	PROC rRUNSIDE1A100()
		MoveJ [[895.91,925.45,959.23],[0.222593,0.0151737,0.948305,-0.225698],[0,-1,0,0],[9E+09,9E+09,9E+09,9E+09,9E+09,9E+09]], vmax, z50, tWeldGun;
		MoveJ [[1169.38,1081.61,325.39],[0.296115,-0.947077,-0.052822,0.112127],[0,-2,0,1],[9E+09,9E+09,9E+09,9E+09,9E+09,9E+09]], vmax, z50, tWeldGun;
		MoveL [[1189.01,1078.57,4.64],[0.333702,-0.921867,0.118424,-0.157418],[0,-2,-1,1],[9E+09,9E+09,9E+09,9E+09,9E+09,9E+09]], v1000, z50, tWeldGun;
		ArcLStart [[1185.61,1080.58,-9.86],[0.333643,-0.921896,0.118528,-0.157299],[0,-2,-1,1],[9E+09,9E+09,9E+09,9E+09,9E+09,9E+09]], v10, seam13, weld13\Weave:=weave1, fine, tWeldGun;
		ArcLEnd [[1153.22,1080.55,-9.89],[0.333626,-0.921901,0.118526,-0.157301],[0,-2,-1,1],[9E+09,9E+09,9E+09,9E+09,9E+09,9E+09]], v10, seam13, weld13\Weave:=weave1, fine, tWeldGun;
		MoveL [[1157.55,1079.96,5.67],[0.333709,-0.921874,0.118398,-0.157383],[0,-2,-1,1],[9E+09,9E+09,9E+09,9E+09,9E+09,9E+09]], vmax, z5, tWeldGun;
		MoveL [[864.56,1073.01,5.26],[0.379695,-0.916748,-0.042496,0.116617],[0,-2,-1,1],[9E+09,9E+09,9E+09,9E+09,9E+09,9E+09]], vmax, z5, tWeldGun;
		ArcLStart [[862.19,1074.19,-3.35],[0.379691,-0.916749,-0.0424859,0.116625],[0,-2,-1,1],[9E+09,9E+09,9E+09,9E+09,9E+09,9E+09]], v10, seam13, weld13\Weave:=weave1, fine, tWeldGun;
		ArcLEnd [[831.24,1074.23,-3.33],[0.379713,-0.916742,-0.0424399,0.116624],[0,-2,-1,1],[9E+09,9E+09,9E+09,9E+09,9E+09,9E+09]], v10, seam13, weld13\Weave:=weave1, fine, tWeldGun;
		MoveL [[834.56,1075.21,12.06],[0.379682,-0.916754,-0.0425092,0.116603],[0,-2,-1,1],[9E+09,9E+09,9E+09,9E+09,9E+09,9E+09]], vmax, z5, tWeldGun;
		MoveL [[172.30,1074.14,5.27],[0.379642,-0.916784,-0.0424626,0.11652],[0,-2,-1,1],[9E+09,9E+09,9E+09,9E+09,9E+09,9E+09]], vmax, z5, tWeldGun;
		ArcLStart [[172.45,1077.16,-3.73],[0.37965,-0.916783,-0.042437,0.116513],[0,-2,-1,1],[9E+09,9E+09,9E+09,9E+09,9E+09,9E+09]], v10, seam13, weld13\Weave:=weave1, fine, tWeldGun;
		ArcLEnd [[141.11,1075.63,-6.35],[0.394237,-0.896713,-0.191368,0.0621412],[0,-2,-1,1],[9E+09,9E+09,9E+09,9E+09,9E+09,9E+09]], v10, seam13, weld13\Weave:=weave1, fine, tWeldGun;
		MoveL [[141.10,1062.84,1.66],[0.394214,-0.896726,-0.191336,0.0621991],[0,-2,-1,1],[9E+09,9E+09,9E+09,9E+09,9E+09,9E+09]], vmax, z5, tWeldGun;
		MoveL [[-144.86,1070.65,3.80],[0.337591,-0.932768,-0.0489574,0.116536],[0,-2,-1,1],[9E+09,9E+09,9E+09,9E+09,9E+09,9E+09]], vmax, z5, tWeldGun;
		ArcLStart [[-144.83,1077.50,-2.20],[0.337605,-0.932765,-0.048953,0.116519],[0,-2,-1,1],[9E+09,9E+09,9E+09,9E+09,9E+09,9E+09]], v10, seam13, weld13\Weave:=weave1, fine, tWeldGun;
		ArcLEnd [[-176.80,1077.27,-2.42],[0.337568,-0.932779,-0.0489017,0.116534],[0,-2,-1,1],[9E+09,9E+09,9E+09,9E+09,9E+09,9E+09]], v10, seam13, weld13\Weave:=weave1, fine, tWeldGun;
		SingArea\Wrist;
		MoveL [[-200.44,1085.42,415.26],[0.379667,-0.916774,-0.042596,0.116465],[0,-2,-1,1],[9E+09,9E+09,9E+09,9E+09,9E+09,9E+09]], vmax, z5, tWeldGun;
		MoveJ [[-173.57,559.75,42.74],[0.145109,0.845875,-0.418866,0.296634],[1,0,-1,0],[9E+09,9E+09,9E+09,9E+09,9E+09,9E+09]], vmax, z5, tWeldGun;
		MoveL [[-170.35,568.46,-5.16],[0.145203,0.845842,-0.418973,0.29653],[1,0,-1,0],[9E+09,9E+09,9E+09,9E+09,9E+09,9E+09]], vmax, z5, tWeldGun;
		ArcLStart [[-170.35,561.67,-11.54],[0.145203,0.845851,-0.418953,0.296532],[1,0,-1,0],[9E+09,9E+09,9E+09,9E+09,9E+09,9E+09]], v10, seam13, weld13\Weave:=weave1, fine, tWeldGun;
		ArcLEnd [[-141.78,561.68,-11.54],[0.145216,0.845844,-0.418977,0.296513],[1,0,-1,0],[9E+09,9E+09,9E+09,9E+09,9E+09,9E+09]], v10, seam13, weld13\Weave:=weave1, fine, tWeldGun;
		MoveL [[-135.50,566.77,5.60],[0.145085,0.84588,-0.41892,0.296555],[1,0,-1,0],[9E+09,9E+09,9E+09,9E+09,9E+09,9E+09]], vmax, z5, tWeldGun;
		MoveL [[151.70,563.89,2.38],[0.145279,0.845821,-0.418979,0.296543],[0,0,-1,0],[9E+09,9E+09,9E+09,9E+09,9E+09,9E+09]], vmax, z5, tWeldGun;
		ArcLStart [[147.91,561.67,-12.61],[0.145298,0.845824,-0.41896,0.296552],[0,0,-1,0],[9E+09,9E+09,9E+09,9E+09,9E+09,9E+09]], v10, seam13, weld13\Weave:=weave1, fine, tWeldGun;
		ArcLEnd [[179.68,561.61,-12.60],[0.145306,0.845823,-0.418965,0.296545],[0,0,-1,0],[9E+09,9E+09,9E+09,9E+09,9E+09,9E+09]], v10, seam13, weld13\Weave:=weave1, fine, tWeldGun;
		MoveL [[179.70,567.65,-1.58],[0.145437,0.845826,-0.418906,0.296553],[0,0,-1,0],[9E+09,9E+09,9E+09,9E+09,9E+09,9E+09]], vmax, z5, tWeldGun;
		MoveL [[838.33,565.65,0.78],[0.145096,0.845788,-0.419047,0.296632],[0,0,-2,0],[9E+09,9E+09,9E+09,9E+09,9E+09,9E+09]], vmax, z5, tWeldGun;
		ArcLStart [[837.91,559.63,-15.44],[0.14512,0.845784,-0.419056,0.29662],[0,0,-2,0],[9E+09,9E+09,9E+09,9E+09,9E+09,9E+09]], v10, seam13, weld13\Weave:=weave1, fine, tWeldGun;
		ArcLEnd [[868.85,559.41,-15.48],[0.145145,0.845802,-0.419023,0.296601],[0,0,-2,0],[9E+09,9E+09,9E+09,9E+09,9E+09,9E+09]], v10, seam13, weld13\Weave:=weave1, fine, tWeldGun;
		MoveL [[869.08,565.56,-7.05],[0.145032,0.845778,-0.419043,0.296696],[0,0,-2,0],[9E+09,9E+09,9E+09,9E+09,9E+09,9E+09]], vmax, z5, tWeldGun;
		MoveL [[1154.26,567.31,-2.43],[0.145055,0.845814,-0.419044,0.296583],[0,0,-2,0],[9E+09,9E+09,9E+09,9E+09,9E+09,9E+09]], vmax, z5, tWeldGun;
		ArcLStart [[1154.25,559.10,-16.64],[0.145066,0.845816,-0.419041,0.296576],[0,0,-2,0],[9E+09,9E+09,9E+09,9E+09,9E+09,9E+09]], v10, seam13, weld13\Weave:=weave1, fine, tWeldGun;
		ArcLEnd [[1186.24,558.29,-16.04],[0.145087,0.845809,-0.419057,0.296562],[0,0,-2,0],[9E+09,9E+09,9E+09,9E+09,9E+09,9E+09]], v10, seam13, weld13\Weave:=weave1, fine, tWeldGun;
		MoveL [[1189.43,560.09,663.81],[0.145007,0.845796,-0.418995,0.296726],[0,0,-2,0],[9E+09,9E+09,9E+09,9E+09,9E+09,9E+09]], vmax, z5, tWeldGun;
		MoveJ [[-229.23,1115.81,554.88],[0.237488,0.691166,-0.628837,0.265431],[1,-1,-4,0],[9E+09,9E+09,9E+09,9E+09,9E+09,9E+09]], vmax, z5, tWeldGun;
		MoveL [[-412.06,717.19,27.71],[0.270403,0.66951,-0.638814,0.265624],[1,0,-4,0],[9E+09,9E+09,9E+09,9E+09,9E+09,9E+09]], vmax, z5, tWeldGun;
		MoveL [[-413.84,720.92,-0.46],[0.249904,0.677081,-0.652542,0.230865],[1,-1,-4,0],[9E+09,9E+09,9E+09,9E+09,9E+09,9E+09]], vmax, z5, tWeldGun;
		ArcLStart [[-413.85,715.51,-6.45],[0.249932,0.67707,-0.652544,0.230859],[1,-1,-4,0],[9E+09,9E+09,9E+09,9E+09,9E+09,9E+09]], v5, seam13, weld13\Weave:=weave1, fine, tWeldGun;
		ArcLEnd [[-433.02,715.70,-6.65],[0.249921,0.677092,-0.652516,0.230888],[1,-1,-4,0],[9E+09,9E+09,9E+09,9E+09,9E+09,9E+09]], v5, seam13, weld13\Weave:=weave1, fine, tWeldGun;
		MoveL [[-433.02,721.69,79.27],[0.249938,0.677071,-0.652532,0.230886],[1,-1,-4,0],[9E+09,9E+09,9E+09,9E+09,9E+09,9E+09]], vmax, z5, tWeldGun;
		MoveL [[-1100.50,721.09,94.11],[0.270393,0.669535,-0.638788,0.265635],[1,-1,-4,0],[9E+09,9E+09,9E+09,9E+09,9E+09,9E+09]], vmax, z5, tWeldGun;
		MoveL [[-1103.19,722.45,8.00],[0.239603,0.681202,-0.652992,0.228379],[1,-1,-4,0],[9E+09,9E+09,9E+09,9E+09,9E+09,9E+09]], vmax, z5, tWeldGun;
		ArcLStart [[-1103.19,713.56,-5.56],[0.239599,0.681202,-0.652993,0.228381],[1,-1,-4,0],[9E+09,9E+09,9E+09,9E+09,9E+09,9E+09]], v5, seam13, weld13\Weave:=weave1, fine, tWeldGun;
		ArcLEnd [[-1123.14,713.55,-4.77],[0.239595,0.681192,-0.652991,0.228416],[1,-1,-4,0],[9E+09,9E+09,9E+09,9E+09,9E+09,9E+09]], v5, seam13, weld13\Weave:=weave1, fine, tWeldGun;
		MoveL [[-1124.97,712.38,115.49],[0.270384,0.669531,-0.638781,0.26567],[1,-1,-4,0],[9E+09,9E+09,9E+09,9E+09,9E+09,9E+09]], vmax, z5, tWeldGun;
		MoveJ [[-1119.62,941.62,98.59],[0.263153,-0.665669,-0.65042,-0.254146],[1,0,-2,0],[9E+09,9E+09,9E+09,9E+09,9E+09,9E+09]], vmax, z5, tWeldGun;
		MoveL [[-1103.53,941.47,2.67],[0.263185,-0.665692,-0.650383,-0.254147],[1,0,-2,0],[9E+09,9E+09,9E+09,9E+09,9E+09,9E+09]], vmax, z5, tWeldGun;
		ArcLStart [[-1102.50,948.16,-6.90],[0.245378,-0.666002,-0.671984,-0.211351],[1,0,-2,0],[9E+09,9E+09,9E+09,9E+09,9E+09,9E+09]], v5, seam13, weld13\Weave:=weave1, fine, tWeldGun;
		ArcL [[-1124.20,945.08,-8.53],[0.241268,-0.666756,-0.672776,-0.211185],[1,0,-2,0],[9E+09,9E+09,9E+09,9E+09,9E+09,9E+09]], v5, seam13, weld13\Weave:=weave1, z10, tWeldGun;
		ArcLEnd [[-1132.51,978.64,-7.54],[0.0250689,0.926224,0.0082503,0.376049],[1,0,-1,0],[9E+09,9E+09,9E+09,9E+09,9E+09,9E+09]], v5, seam13, weld13\Weave:=weave1, fine, tWeldGun;
		MoveL [[-1148.62,985.17,63.09],[0.0198579,0.898733,0.00249179,0.438039],[1,-1,-1,0],[9E+09,9E+09,9E+09,9E+09,9E+09,9E+09]], vmax, z5, tWeldGun;
		MoveL [[-1199.14,1157.80,50.93],[0.0198608,0.898743,0.00250084,0.43802],[1,-1,-1,0],[9E+09,9E+09,9E+09,9E+09,9E+09,9E+09]], vmax, z5, tWeldGun;
		MoveL [[-1195.49,1156.64,0.22],[0.0202314,0.914596,0.00160063,0.403859],[1,0,-1,0],[9E+09,9E+09,9E+09,9E+09,9E+09,9E+09]], vmax, z5, tWeldGun;
		ArcLStart [[-1192.13,1157.24,-7.56],[0.0202377,0.91461,0.00159549,0.403829],[1,0,-1,0],[9E+09,9E+09,9E+09,9E+09,9E+09,9E+09]], v5, seam13, weld13\Weave:=weave1, fine, tWeldGun;
		ArcL [[-1195.11,1177.16,-6.96],[0.0243873,0.92589,-0.000794778,0.377005],[1,0,-1,0],[9E+09,9E+09,9E+09,9E+09,9E+09,9E+09]], v5, seam13, weld13\Weave:=weave1, z10, tWeldGun;
		ArcLEnd [[-1166.64,1194.35,-4.47],[0.234917,0.673253,-0.666667,0.217024],[1,-1,0,0],[9E+09,9E+09,9E+09,9E+09,9E+09,9E+09]], v5, seam13, weld13\Weave:=weave1, fine, tWeldGun;
		MoveL [[-1164.13,1200.44,93.33],[0.251271,0.657126,-0.66952,0.23831],[1,-1,0,0],[9E+09,9E+09,9E+09,9E+09,9E+09,9E+09]], vmax, z5, tWeldGun;
		MoveJ [[-1176.39,1428.24,109.35],[0.303454,-0.641239,-0.63752,-0.300495],[1,-1,2,0],[9E+09,9E+09,9E+09,9E+09,9E+09,9E+09]], vmax, z5, tWeldGun;
		MoveL [[-1186.42,1420.24,9.09],[0.262683,-0.660481,-0.654281,-0.258224],[1,0,2,0],[9E+09,9E+09,9E+09,9E+09,9E+09,9E+09]], vmax, z5, tWeldGun;
		ArcLStart [[-1183.89,1427.01,-5.32],[0.262685,-0.660493,-0.654268,-0.258224],[1,0,2,0],[9E+09,9E+09,9E+09,9E+09,9E+09,9E+09]], v30, seam13, weld13\Weave:=weave1, fine, tWeldGun;
		ArcLEnd [[-1164.71,1427.19,-6.55],[0.262711,-0.66047,-0.654286,-0.258211],[1,0,2,0],[9E+09,9E+09,9E+09,9E+09,9E+09,9E+09]], v5, seam13, weld13\Weave:=weave1, fine, tWeldGun;
		MoveL [[-1165.10,1427.68,74.68],[0.262682,-0.660472,-0.654289,-0.258226],[1,0,2,0],[9E+09,9E+09,9E+09,9E+09,9E+09,9E+09]], vmax, z5, tWeldGun;
		MoveL [[-495.20,1424.53,122.41],[0.28862,-0.64963,-0.643265,-0.284411],[1,-1,2,0],[9E+09,9E+09,9E+09,9E+09,9E+09,9E+09]], vmax, z5, tWeldGun;
		MoveL [[-492.11,1424.64,-4.56],[0.230632,-0.671635,-0.668577,-0.220728],[1,0,2,0],[9E+09,9E+09,9E+09,9E+09,9E+09,9E+09]], vmax, z5, tWeldGun;
		ArcLStart [[-494.82,1430.84,-11.36],[0.230629,-0.671668,-0.668546,-0.220726],[1,0,2,0],[9E+09,9E+09,9E+09,9E+09,9E+09,9E+09]], v5, seam13, weld13\Weave:=weave1, fine, tWeldGun;
		ArcLEnd [[-475.00,1430.64,-11.57],[0.230621,-0.671683,-0.668534,-0.220724],[1,0,2,0],[9E+09,9E+09,9E+09,9E+09,9E+09,9E+09]], v5, seam13, weld13\Weave:=weave1, fine, tWeldGun;
		MoveL [[-474.63,1411.30,125.45],[0.288602,-0.649679,-0.643225,-0.284408],[1,-1,2,0],[9E+09,9E+09,9E+09,9E+09,9E+09,9E+09]], vmax, z5, tWeldGun;
		MoveJ [[-479.04,1241.31,118.19],[0.268582,0.650118,-0.664304,0.252806],[1,-1,0,0],[9E+09,9E+09,9E+09,9E+09,9E+09,9E+09]], vmax, z5, tWeldGun;
		MoveL [[-495.83,1201.80,-1.90],[0.268594,0.650121,-0.6643,0.252797],[1,-1,0,0],[9E+09,9E+09,9E+09,9E+09,9E+09,9E+09]], vmax, z5, tWeldGun;
		ArcLStart [[-494.84,1196.21,-9.49],[0.268603,0.650127,-0.664292,0.252793],[1,-1,0,0],[9E+09,9E+09,9E+09,9E+09,9E+09,9E+09]], v5, seam13, weld13\Weave:=weave1, fine, tWeldGun;
		ArcL [[-476.48,1196.50,-9.26],[0.268632,0.650097,-0.664312,0.252787],[1,-1,0,0],[9E+09,9E+09,9E+09,9E+09,9E+09,9E+09]], v5, seam13, weld13\Weave:=weave1, z10, tWeldGun;
		ArcLEnd [[-465.51,1166.36,-12.09],[0.390509,0.0535053,-0.919043,-0.000194166],[1,-1,1,0],[9E+09,9E+09,9E+09,9E+09,9E+09,9E+09]], v5, seam13, weld13\Weave:=weave1, fine, tWeldGun;
		MoveL [[-435.96,1164.94,59.58],[0.390502,0.0535497,-0.919044,-0.000186584],[1,-1,1,0],[9E+09,9E+09,9E+09,9E+09,9E+09,9E+09]], vmax, z5, tWeldGun;
		MoveL [[-398.53,986.99,7.96],[0.390518,0.0535228,-0.919039,-0.00018247],[1,-1,1,0],[9E+09,9E+09,9E+09,9E+09,9E+09,9E+09]], vmax, z5, tWeldGun;
		ArcLStart [[-404.11,986.56,-9.77],[0.390535,0.0535541,-0.919029,-0.000151074],[1,-1,1,0],[9E+09,9E+09,9E+09,9E+09,9E+09,9E+09]], v20, seam13, weld13\Weave:=weave1, fine, tWeldGun;
		ArcL [[-404.10,964.74,-9.51],[0.390566,0.0535448,-0.919017,-0.000185269],[1,-1,1,0],[9E+09,9E+09,9E+09,9E+09,9E+09,9E+09]], v5, seam13, weld13\Weave:=weave1, z10, tWeldGun;
		ArcLEnd [[-428.88,950.30,-8.06],[0.237036,-0.623338,-0.70044,-0.254259],[1,-1,2,0],[9E+09,9E+09,9E+09,9E+09,9E+09,9E+09]], v5, seam13, weld13\Weave:=weave1, fine, tWeldGun;
		MoveL [[-432.86,900.19,113.28],[0.289357,-0.647919,-0.645007,-0.283619],[1,-1,2,0],[9E+09,9E+09,9E+09,9E+09,9E+09,9E+09]], vmax, z5, tWeldGun;
		MoveJ [[276.57,1109.67,795.31],[0.28935,-0.647904,-0.645024,-0.283623],[0,0,1,0],[9E+09,9E+09,9E+09,9E+09,9E+09,9E+09]], vmax, z5, tWeldGun;
	ENDPROC
	PROC ProSkid200()
		MoveJ pSafeS1, vmax, fine, tWeldGun;
		MoveL [[-234.96,1621.92,-8.21],[0.194298,-0.276185,-0.910115,-0.24013],[1,-1,1,0],[9E+09,9E+09,9E+09,9E+09,9E+09,9E+09]], vmax, z50, tWeldGun;
		SingArea\Wrist;
		ArcLStart [[-265.19,1628.57,-38.88],[0.243445,-0.67037,-0.655025,-0.249563],[1,0,2,0],[9E+09,9E+09,9E+09,9E+09,9E+09,9E+09]], v40, seam13, weld13, fine, tWeldGun;
		ArcLEnd [[-257.54,1628.57,-38.88],[0.243445,-0.670369,-0.655025,-0.249565],[1,0,2,0],[9E+09,9E+09,9E+09,9E+09,9E+09,9E+09]], v10, seam13, weld13, fine, tWeldGun;
		MoveL [[-258.35,1618.76,-2.87],[0.243441,-0.670362,-0.655032,-0.24957],[1,0,2,0],[9E+09,9E+09,9E+09,9E+09,9E+09,9E+09]], vmax, z20, tWeldGun;
		MoveJ [[-252.87,717.22,166.31],[0.308554,0.634187,-0.646071,0.291883],[1,0,0,0],[9E+09,9E+09,9E+09,9E+09,9E+09,9E+09]], vmax, z20, tWeldGun;
		SingArea\Wrist;
		MoveL [[-273.06,697.08,-39.01],[0.289422,0.639754,-0.670959,0.238254],[1,0,0,0],[9E+09,9E+09,9E+09,9E+09,9E+09,9E+09]], vmax, z20, tWeldGun;
		ArcLStart [[-273.06,687.07,-45.02],[0.289425,0.639748,-0.670962,0.238258],[1,0,0,0],[9E+09,9E+09,9E+09,9E+09,9E+09,9E+09]], v10, seam13, weld13, fine, tWeldGun;
		ArcLEnd [[-266.46,687.08,-45.02],[0.289425,0.63975,-0.67096,0.238257],[1,0,0,0],[9E+09,9E+09,9E+09,9E+09,9E+09,9E+09]], v10, seam13, weld13, fine, tWeldGun;
		MoveL [[-265.17,697.65,3.08],[0.289425,0.639755,-0.670954,0.238258],[1,0,0,0],[9E+09,9E+09,9E+09,9E+09,9E+09,9E+09]], vmax, z20, tWeldGun;
		MoveJ [[1363.12,672.47,163.81],[0.230647,0.704641,-0.28697,0.606574],[0,-1,-1,0],[9E+09,9E+09,9E+09,9E+09,9E+09,9E+09]], vmax, z20, tWeldGun;
		MoveL [[1363.13,672.48,-59.34],[0.230635,0.704646,-0.28697,0.606573],[0,-1,-1,0],[9E+09,9E+09,9E+09,9E+09,9E+09,9E+09]], vmax, z20, tWeldGun;
		ArcLStart [[1395.10,665.67,-59.36],[0.230647,0.704646,-0.286968,0.606569],[0,-1,-1,0],[9E+09,9E+09,9E+09,9E+09,9E+09,9E+09]], v10, seam13, weld13, fine, tWeldGun;
		ArcLEnd [[1393.21,666.82,-105.76],[0.230653,0.704647,-0.286991,0.606554],[0,-1,-1,0],[9E+09,9E+09,9E+09,9E+09,9E+09,9E+09]], v10, seam13, weld13, fine, tWeldGun;
		MoveL [[1360.51,678.95,-105.76],[0.230657,0.704646,-0.286998,0.60655],[0,-1,-1,0],[9E+09,9E+09,9E+09,9E+09,9E+09,9E+09]], vmax, z20, tWeldGun;
		MoveJ [[1360.48,679.11,200.26],[0.227916,0.703475,-0.290109,0.607465],[0,-1,-1,0],[9E+09,9E+09,9E+09,9E+09,9E+09,9E+09]], vmax, z20, tWeldGun;
		MoveJ [[1372.60,1612.03,89.61],[0.238536,-0.688587,-0.26592,-0.631059],[0,-1,-2,0],[9E+09,9E+09,9E+09,9E+09,9E+09,9E+09]], vmax, z20, tWeldGun;
		MoveL [[1372.62,1612.07,-51.09],[0.238534,-0.68856,-0.265944,-0.631079],[0,-1,-2,0],[9E+09,9E+09,9E+09,9E+09,9E+09,9E+09]], vmax, z20, tWeldGun;
		ArcLStart [[1403.05,1622.70,-51.46],[0.238475,-0.688587,-0.265917,-0.631084],[0,-1,-2,0],[9E+09,9E+09,9E+09,9E+09,9E+09,9E+09]], v10, seam13, weld13, fine, tWeldGun;
		ArcLEnd [[1401.72,1623.96,-98.89],[0.23847,-0.688542,-0.266036,-0.631085],[0,-1,-2,0],[9E+09,9E+09,9E+09,9E+09,9E+09,9E+09]], v10, seam13, weld13, fine, tWeldGun;
		MoveL [[1350.78,1600.25,-98.94],[0.23849,-0.68857,-0.265983,-0.631068],[0,-1,-2,0],[9E+09,9E+09,9E+09,9E+09,9E+09,9E+09]], vmax, z20, tWeldGun;
		MoveL [[1286.32,1556.33,142.30],[0.238485,-0.688572,-0.265997,-0.631063],[0,-1,-2,0],[9E+09,9E+09,9E+09,9E+09,9E+09,9E+09]], vmax, z20, tWeldGun;
		MoveJ [[1024.21,1614.84,123.96],[0.621106,-0.285749,-0.670591,-0.287895],[0,0,0,0],[9E+09,9E+09,9E+09,9E+09,9E+09,9E+09]], vmax, z20, tWeldGun;
		MoveL [[1024.31,1614.97,-44.55],[0.621177,-0.285699,-0.670494,-0.288017],[0,0,0,0],[9E+09,9E+09,9E+09,9E+09,9E+09,9E+09]], vmax, z20, tWeldGun;
		ArcLStart [[986.78,1630.52,-48.85],[0.621168,-0.285689,-0.670501,-0.28803],[0,0,0,0],[9E+09,9E+09,9E+09,9E+09,9E+09,9E+09]], v10, seam13, weld13, fine, tWeldGun;
		ArcLEnd [[989.07,1629.80,-94.04],[0.621174,-0.285677,-0.670503,-0.288024],[0,0,0,0],[9E+09,9E+09,9E+09,9E+09,9E+09,9E+09]], v10, seam13, weld13, fine, tWeldGun;
		MoveL [[1031.38,1620.08,-94.06],[0.621173,-0.285694,-0.670496,-0.288025],[0,0,0,0],[9E+09,9E+09,9E+09,9E+09,9E+09,9E+09]], vmax, z20, tWeldGun;
		MoveL [[1050.77,1575.36,86.67],[0.621174,-0.285691,-0.670496,-0.288026],[0,0,0,0],[9E+09,9E+09,9E+09,9E+09,9E+09,9E+09]], vmax, z20, tWeldGun;
		MoveJ [[1013.51,687.74,143.37],[0.59856,0.318284,-0.67023,0.302017],[0,-1,-1,0],[9E+09,9E+09,9E+09,9E+09,9E+09,9E+09]], vmax, z20, tWeldGun;
		MoveL [[1013.45,687.71,-58.15],[0.598615,0.318227,-0.670196,0.302042],[0,-1,-1,0],[9E+09,9E+09,9E+09,9E+09,9E+09,9E+09]], vmax, z20, tWeldGun;
		ArcLStart [[981.75,669.03,-58.14],[0.598616,0.318216,-0.6702,0.302041],[0,-1,-1,0],[9E+09,9E+09,9E+09,9E+09,9E+09,9E+09]], v10, seam13, weld13, fine, tWeldGun;
		ArcLEnd [[981.75,669.03,-102.94],[0.598614,0.318211,-0.670206,0.302041],[0,-1,-1,0],[9E+09,9E+09,9E+09,9E+09,9E+09,9E+09]], v10, seam13, weld13, fine, tWeldGun;
		MoveL [[1021.06,692.65,-100.54],[0.598619,0.318178,-0.670217,0.30204],[0,-1,-1,0],[9E+09,9E+09,9E+09,9E+09,9E+09,9E+09]], vmax, z20, tWeldGun;
		MoveL [[1021.06,692.65,172.93],[0.598621,0.318175,-0.670218,0.302038],[0,-1,-1,0],[9E+09,9E+09,9E+09,9E+09,9E+09,9E+09]], vmax, z20, tWeldGun;
		MoveJ [[962.66,684.38,264.32],[0.236784,0.681997,-0.2918,0.627429],[0,1,1,1],[9E+09,9E+09,9E+09,9E+09,9E+09,9E+09]], vmax, z20, tWeldGun;
		MoveL [[962.64,684.38,-48.75],[0.236792,0.682002,-0.291815,0.627413],[0,1,1,1],[9E+09,9E+09,9E+09,9E+09,9E+09,9E+09]], vmax, z20, tWeldGun;
		ArcLStart [[980.94,668.93,-48.75],[0.236782,0.682005,-0.291808,0.627418],[0,1,1,1],[9E+09,9E+09,9E+09,9E+09,9E+09,9E+09]], v10, seam13, weld13, fine, tWeldGun;
		ArcLEnd [[980.92,669.75,-104.66],[0.236799,0.682008,-0.291831,0.627396],[0,1,1,1],[9E+09,9E+09,9E+09,9E+09,9E+09,9E+09]], v10, seam13, weld13, fine, tWeldGun;
		MoveL [[948.38,696.75,-105.45],[0.234731,0.68317,-0.291592,0.62702],[0,1,1,1],[9E+09,9E+09,9E+09,9E+09,9E+09,9E+09]], vmax, z20, tWeldGun;
		MoveL [[948.40,696.76,143.62],[0.234722,0.683169,-0.291572,0.627035],[0,1,1,1],[9E+09,9E+09,9E+09,9E+09,9E+09,9E+09]], vmax, z20, tWeldGun;
		MoveJ [[975.43,1612.68,308.57],[0.225877,-0.689512,-0.28382,-0.626896],[0,1,0,1],[9E+09,9E+09,9E+09,9E+09,9E+09,9E+09]], vmax, z20, tWeldGun;
		MoveL [[975.55,1612.35,-40.05],[0.22557,-0.689612,-0.283854,-0.626882],[0,0,1,1],[9E+09,9E+09,9E+09,9E+09,9E+09,9E+09]], vmax, z20, tWeldGun;
		ArcLStart [[989.75,1627.18,-40.10],[0.225683,-0.689679,-0.283801,-0.626791],[0,1,1,1],[9E+09,9E+09,9E+09,9E+09,9E+09,9E+09]], v10, seam13, weld13, fine, tWeldGun;
		ArcLEnd [[988.02,1626.51,-103.36],[0.218861,-0.704472,-0.289009,-0.610159],[0,1,1,1],[9E+09,9E+09,9E+09,9E+09,9E+09,9E+09]], v10, seam13, weld13, fine, tWeldGun;
		MoveL [[969.19,1616.42,-103.36],[0.21886,-0.704489,-0.288978,-0.610154],[0,1,1,1],[9E+09,9E+09,9E+09,9E+09,9E+09,9E+09]], vmax, z20, tWeldGun;
		MoveL [[972.04,1615.87,168.33],[0.225681,-0.689708,-0.283758,-0.62678],[0,1,0,1],[9E+09,9E+09,9E+09,9E+09,9E+09,9E+09]], vmax, z20, tWeldGun;
		MoveJ [[748.32,1594.78,-28.74],[0.231269,-0.620927,-0.702805,-0.258902],[0,1,-1,1],[9E+09,9E+09,9E+09,9E+09,9E+09,9E+09]], vmax, z20, tWeldGun;
		MoveL [[748.32,1618.27,-62.58],[0.231267,-0.620927,-0.702807,-0.258898],[0,1,-1,1],[9E+09,9E+09,9E+09,9E+09,9E+09,9E+09]], vmax, z20, tWeldGun;
		ArcLStart [[748.35,1622.75,-67.83],[0.23126,-0.620915,-0.702812,-0.25892],[0,1,-1,1],[9E+09,9E+09,9E+09,9E+09,9E+09,9E+09]], v10, seam13, weld13, fine, tWeldGun;
		ArcLEnd [[720.93,1622.75,-67.82],[0.231262,-0.620925,-0.702803,-0.258918],[0,1,-1,1],[9E+09,9E+09,9E+09,9E+09,9E+09,9E+09]], v10, seam13, weld13, fine, tWeldGun;
		MoveL [[683.13,1622.94,-67.84],[0.231262,-0.620938,-0.702794,-0.258913],[0,1,-1,1],[9E+09,9E+09,9E+09,9E+09,9E+09,9E+09]], vmax, z20, tWeldGun;
		ArcLStart [[681.00,1622.93,-67.87],[0.231258,-0.62095,-0.702784,-0.258913],[0,1,-1,1],[9E+09,9E+09,9E+09,9E+09,9E+09,9E+09]], v10, seam13, weld13, fine, tWeldGun;
		ArcLEnd [[654.73,1623.14,-67.84],[0.231266,-0.620945,-0.702787,-0.258912],[0,1,-1,1],[9E+09,9E+09,9E+09,9E+09,9E+09,9E+09]], v10, seam13, weld13, fine, tWeldGun;
		MoveL [[654.72,1619.33,-13.30],[0.231269,-0.620959,-0.702776,-0.258903],[0,1,-1,1],[9E+09,9E+09,9E+09,9E+09,9E+09,9E+09]], vmax, z20, tWeldGun;
		MoveJ [[37.05,1622.28,-7.90],[0.231269,-0.620971,-0.702762,-0.258912],[1,1,-1,1],[9E+09,9E+09,9E+09,9E+09,9E+09,9E+09]], vmax, z20, tWeldGun;
		MoveL [[37.06,1622.28,-65.61],[0.231267,-0.620964,-0.702769,-0.258912],[1,1,-1,1],[9E+09,9E+09,9E+09,9E+09,9E+09,9E+09]], vmax, z20, tWeldGun;
		ArcLStart [[37.05,1628.08,-65.61],[0.231271,-0.620973,-0.702759,-0.258914],[1,1,-1,1],[9E+09,9E+09,9E+09,9E+09,9E+09,9E+09]], v10, seam13, weld13, fine, tWeldGun;
		ArcLEnd [[7.65,1628.68,-65.60],[0.231271,-0.620979,-0.702755,-0.258912],[1,1,-1,1],[9E+09,9E+09,9E+09,9E+09,9E+09,9E+09]], v10, seam13, weld13, fine, tWeldGun;
		MoveL [[-27.35,1629.08,-65.60],[0.231271,-0.620982,-0.702752,-0.258911],[1,1,0,1],[9E+09,9E+09,9E+09,9E+09,9E+09,9E+09]], vmax, z20, tWeldGun;
		ArcLStart [[-31.75,1629.08,-65.60],[0.231272,-0.620988,-0.702747,-0.258912],[1,1,0,1],[9E+09,9E+09,9E+09,9E+09,9E+09,9E+09]], v10, seam13, weld13, fine, tWeldGun;
		ArcLEnd [[-60.36,1629.07,-65.63],[0.231269,-0.621009,-0.70273,-0.258909],[1,1,0,1],[9E+09,9E+09,9E+09,9E+09,9E+09,9E+09]], v10, seam13, weld13, fine, tWeldGun;
		MoveL [[-63.19,1451.21,44.92],[0.231265,-0.62101,-0.702733,-0.258902],[1,1,0,1],[9E+09,9E+09,9E+09,9E+09,9E+09,9E+09]], vmax, z20, tWeldGun;
		SingArea\Wrist;
		MoveJ [[-220.42,1456.39,142.20],[0.365991,-0.606888,-0.673424,-0.210328],[1,0,1,0],[9E+09,9E+09,9E+09,9E+09,9E+09,9E+09]], vmax, z20, tWeldGun;
		MoveL [[-219.91,1623.63,-54.86],[0.365978,-0.606856,-0.673457,-0.210339],[1,0,1,0],[9E+09,9E+09,9E+09,9E+09,9E+09,9E+09]], vmax, z20, tWeldGun;
		ArcLStart [[-219.83,1630.03,-63.47],[0.36598,-0.606851,-0.67346,-0.21034],[1,0,1,0],[9E+09,9E+09,9E+09,9E+09,9E+09,9E+09]], v10, seam13, weld13, fine, tWeldGun;
		ArcLEnd [[-233.82,1630.03,-62.87],[0.365977,-0.606844,-0.673467,-0.210341],[1,0,1,0],[9E+09,9E+09,9E+09,9E+09,9E+09,9E+09]], v10, seam13, weld13, fine, tWeldGun;
		MoveL [[-229.83,1622.04,44.03],[0.365923,-0.606933,-0.673436,-0.21028],[1,0,1,0],[9E+09,9E+09,9E+09,9E+09,9E+09,9E+09]], vmax, z20, tWeldGun;
		MoveJ [[-238.42,695.07,107.36],[0.416175,0.412803,-0.798145,0.139133],[1,0,0,0],[9E+09,9E+09,9E+09,9E+09,9E+09,9E+09]], vmax, z20, tWeldGun;
		MoveL [[-238.43,695.09,-59.53],[0.416176,0.412786,-0.798155,0.139122],[1,0,0,0],[9E+09,9E+09,9E+09,9E+09,9E+09,9E+09]], vmax, z20, tWeldGun;
		ArcLStart [[-240.41,687.67,-69.36],[0.416165,0.412798,-0.798152,0.139137],[1,0,0,0],[9E+09,9E+09,9E+09,9E+09,9E+09,9E+09]], v10, seam13, weld13, fine, tWeldGun;
		ArcLEnd [[-225.81,687.67,-69.75],[0.416158,0.41281,-0.798148,0.139143],[1,0,0,0],[9E+09,9E+09,9E+09,9E+09,9E+09,9E+09]], v10, seam13, weld13, fine, tWeldGun;
		MoveL [[-226.30,704.95,-17.45],[0.416163,0.412818,-0.79814,0.139151],[1,0,0,0],[9E+09,9E+09,9E+09,9E+09,9E+09,9E+09]], vmax, z20, tWeldGun;
		MoveJ [[-68.54,708.92,-17.46],[0.33715,0.641758,-0.612556,0.315044],[1,0,-1,0],[9E+09,9E+09,9E+09,9E+09,9E+09,9E+09]], vmax, z20, tWeldGun;
		MoveL [[-69.37,694.59,-61.82],[0.293998,0.661849,-0.635411,0.267907],[1,0,-1,0],[9E+09,9E+09,9E+09,9E+09,9E+09,9E+09]], vmax, z20, tWeldGun;
		ArcLStart [[-69.36,687.96,-70.31],[0.294028,0.661818,-0.635424,0.26792],[1,0,-1,0],[9E+09,9E+09,9E+09,9E+09,9E+09,9E+09]], v10, seam13, weld13, fine, tWeldGun;
		ArcLEnd [[-41.96,687.95,-70.52],[0.29404,0.66181,-0.635427,0.267921],[1,0,-1,0],[9E+09,9E+09,9E+09,9E+09,9E+09,9E+09]], v10, seam13, weld13, fine, tWeldGun;
		MoveL [[-6.97,687.95,-70.51],[0.294043,0.661806,-0.635431,0.267916],[0,0,-1,0],[9E+09,9E+09,9E+09,9E+09,9E+09,9E+09]], vmax, z20, tWeldGun;
		ArcLStart [[-6.96,687.54,-70.52],[0.294045,0.661806,-0.635429,0.267919],[0,0,-1,0],[9E+09,9E+09,9E+09,9E+09,9E+09,9E+09]], v10, seam13, weld13, fine, tWeldGun;
		ArcLEnd [[21.80,686.99,-70.51],[0.294054,0.661794,-0.635442,0.267908],[0,0,-1,0],[9E+09,9E+09,9E+09,9E+09,9E+09,9E+09]], v10, seam13, weld13, fine, tWeldGun;
		MoveL [[21.80,693.66,-56.32],[0.294011,0.661823,-0.635446,0.267875],[0,0,-1,0],[9E+09,9E+09,9E+09,9E+09,9E+09,9E+09]], vmax, z20, tWeldGun;
		MoveL [[644.60,694.09,-38.11],[0.29406,0.661788,-0.635447,0.267906],[0,0,-1,0],[9E+09,9E+09,9E+09,9E+09,9E+09,9E+09]], vmax, z20, tWeldGun;
		ArcLStart [[644.53,682.78,-73.42],[0.294076,0.661755,-0.635493,0.267859],[0,0,-1,0],[9E+09,9E+09,9E+09,9E+09,9E+09,9E+09]], v40, seam13, weld13, fine, tWeldGun;
		ArcLEnd [[667.66,682.46,-73.44],[0.294106,0.661729,-0.635513,0.267845],[0,0,-1,0],[9E+09,9E+09,9E+09,9E+09,9E+09,9E+09]], v10, seam13, weld13, fine, tWeldGun;
		MoveL [[706.98,682.46,-73.44],[0.294117,0.661731,-0.635507,0.267842],[0,0,-1,0],[9E+09,9E+09,9E+09,9E+09,9E+09,9E+09]], vmax, z20, tWeldGun;
		ArcLStart [[706.98,682.46,-73.44],[0.294117,0.66173,-0.635507,0.267841],[0,0,-1,0],[9E+09,9E+09,9E+09,9E+09,9E+09,9E+09]], v10, seam13, weld13, fine, tWeldGun;
		ArcLEnd [[732.78,682.64,-73.45],[0.294116,0.66175,-0.635481,0.267856],[0,0,-1,0],[9E+09,9E+09,9E+09,9E+09,9E+09,9E+09]], v10, seam13, weld13, fine, tWeldGun;
		MoveL [[743.36,710.11,-13.87],[0.294132,0.661743,-0.635486,0.267845],[0,0,-1,0],[9E+09,9E+09,9E+09,9E+09,9E+09,9E+09]], vmax, z20, tWeldGun;
		MoveJ [[766.73,689.09,12.78],[0.426939,0.266425,-0.809663,0.301972],[0,-1,0,0],[9E+09,9E+09,9E+09,9E+09,9E+09,9E+09]], vmax, z20, tWeldGun;
		MoveL [[766.72,689.01,-73.04],[0.426946,0.266425,-0.809635,0.302037],[0,-1,0,0],[9E+09,9E+09,9E+09,9E+09,9E+09,9E+09]], vmax, z20, tWeldGun;
		ArcLStart [[753.37,674.21,-83.82],[0.426978,0.266403,-0.80963,0.302027],[0,-1,0,0],[9E+09,9E+09,9E+09,9E+09,9E+09,9E+09]], v10, seam13, weld13, fine, tWeldGun;
		ArcLEnd [[753.94,674.20,-111.42],[0.427004,0.266403,-0.809617,0.302024],[0,-1,0,0],[9E+09,9E+09,9E+09,9E+09,9E+09,9E+09]], v10, seam13, weld13, fine, tWeldGun;
		MoveL [[767.24,687.28,-25.85],[0.427002,0.266345,-0.809691,0.301878],[0,-1,0,0],[9E+09,9E+09,9E+09,9E+09,9E+09,9E+09]], vmax, z20, tWeldGun;
		MoveJ [[43.23,696.82,-1.72],[0.42676,0.266354,-0.810055,0.301235],[0,-1,0,0],[9E+09,9E+09,9E+09,9E+09,9E+09,9E+09]], vmax, z20, tWeldGun;
		MoveL [[42.01,683.49,-78.40],[0.427024,0.26632,-0.809694,0.301862],[0,-1,0,0],[9E+09,9E+09,9E+09,9E+09,9E+09,9E+09]], vmax, z20, tWeldGun;
		ArcLStart [[38.82,680.87,-78.40],[0.427033,0.266358,-0.80967,0.301881],[0,-1,0,0],[9E+09,9E+09,9E+09,9E+09,9E+09,9E+09]], v10, seam13, weld13, fine, tWeldGun;
		ArcLEnd [[40.20,680.75,-109.60],[0.427039,0.266382,-0.80967,0.301849],[0,-1,0,0],[9E+09,9E+09,9E+09,9E+09,9E+09,9E+09]], v10, seam13, weld13, fine, tWeldGun;
		MoveL [[56.60,714.15,-11.47],[0.427063,0.266301,-0.809685,0.301848],[0,-1,0,0],[9E+09,9E+09,9E+09,9E+09,9E+09,9E+09]], vmax, z20, tWeldGun;
		MoveJ [[-90.85,716.79,14.15],[0.243321,0.796043,-0.267285,0.485459],[1,-1,-1,0],[9E+09,9E+09,9E+09,9E+09,9E+09,9E+09]], vmax, z20, tWeldGun;
		MoveL [[-92.64,686.16,-78.85],[0.243349,0.796017,-0.267252,0.485505],[1,-1,-1,0],[9E+09,9E+09,9E+09,9E+09,9E+09,9E+09]], vmax, z20, tWeldGun;
		ArcLStart [[-85.54,680.97,-78.85],[0.243338,0.796021,-0.267256,0.485502],[1,-1,-1,0],[9E+09,9E+09,9E+09,9E+09,9E+09,9E+09]], v10, seam13, weld13, fine, tWeldGun;
		ArcLEnd [[-85.54,680.97,-106.06],[0.243338,0.796019,-0.267253,0.485507],[1,-1,-1,0],[9E+09,9E+09,9E+09,9E+09,9E+09,9E+09]], v10, seam13, weld13, fine, tWeldGun;
		MoveL [[-99.62,700.82,-3.32],[0.243332,0.796035,-0.267233,0.485495],[1,-1,-1,0],[9E+09,9E+09,9E+09,9E+09,9E+09,9E+09]], vmax, z20, tWeldGun;
		MoveJ [[622.81,695.86,-3.35],[0.24331,0.796057,-0.26719,0.485493],[0,-1,-1,0],[9E+09,9E+09,9E+09,9E+09,9E+09,9E+09]], vmax, z20, tWeldGun;
		MoveL [[622.81,678.68,-81.59],[0.243312,0.796055,-0.267198,0.485492],[0,-1,-1,0],[9E+09,9E+09,9E+09,9E+09,9E+09,9E+09]], vmax, z20, tWeldGun;
		ArcLStart [[627.79,674.24,-83.40],[0.243343,0.796045,-0.267192,0.485495],[0,-1,-1,0],[9E+09,9E+09,9E+09,9E+09,9E+09,9E+09]], v10, seam13, weld13, fine, tWeldGun;
		ArcLEnd [[626.78,674.63,-109.81],[0.243358,0.796042,-0.267204,0.485485],[0,-1,-1,0],[9E+09,9E+09,9E+09,9E+09,9E+09,9E+09]], v10, seam13, weld13, fine, tWeldGun;
		MoveL [[610.77,692.21,49.90],[0.243321,0.79605,-0.267267,0.485457],[0,-1,-1,0],[9E+09,9E+09,9E+09,9E+09,9E+09,9E+09]], vmax, z20, tWeldGun;
		MoveJ [[622.12,1614.25,159.14],[0.192579,-0.77773,-0.32949,-0.499486],[0,1,0,1],[9E+09,9E+09,9E+09,9E+09,9E+09,9E+09]], vmax, z20, tWeldGun;
		MoveL [[622.15,1614.23,-75.01],[0.192557,-0.777696,-0.329551,-0.499508],[0,1,0,1],[9E+09,9E+09,9E+09,9E+09,9E+09,9E+09]], vmax, z20, tWeldGun;
		ArcLStart [[640.60,1627.79,-79.81],[0.192567,-0.777665,-0.329604,-0.499517],[0,1,0,1],[9E+09,9E+09,9E+09,9E+09,9E+09,9E+09]], v10, seam13, weld13, fine, tWeldGun;
		ArcLEnd [[640.40,1627.75,-105.01],[0.19256,-0.777691,-0.32956,-0.499508],[0,1,0,1],[9E+09,9E+09,9E+09,9E+09,9E+09,9E+09]], v10, seam13, weld13, fine, tWeldGun;
		MoveL [[622.01,1617.53,-16.15],[0.192549,-0.777705,-0.329542,-0.499501],[0,1,0,1],[9E+09,9E+09,9E+09,9E+09,9E+09,9E+09]], vmax, z20, tWeldGun;
		MoveJ [[-74.83,1621.54,-16.16],[0.19255,-0.777728,-0.329501,-0.499493],[1,1,0,1],[9E+09,9E+09,9E+09,9E+09,9E+09,9E+09]], vmax, z20, tWeldGun;
		MoveL [[-74.84,1632.22,-76.43],[0.192546,-0.777738,-0.329487,-0.499489],[1,1,0,1],[9E+09,9E+09,9E+09,9E+09,9E+09,9E+09]], vmax, z20, tWeldGun;
		ArcLStart [[-72.04,1634.00,-74.85],[0.192535,-0.777754,-0.329462,-0.499484],[1,1,0,1],[9E+09,9E+09,9E+09,9E+09,9E+09,9E+09]], v10, seam13, weld13, fine, tWeldGun;
		ArcLEnd [[-72.05,1633.99,-104.27],[0.19253,-0.777762,-0.329453,-0.49948],[1,1,0,1],[9E+09,9E+09,9E+09,9E+09,9E+09,9E+09]], v10, seam13, weld13, fine, tWeldGun;
		MoveL [[-101.85,1558.57,140.36],[0.192608,-0.777808,-0.329372,-0.499431],[1,1,0,1],[9E+09,9E+09,9E+09,9E+09,9E+09,9E+09]], vmax, z20, tWeldGun;
		MoveJ [[102.30,1319.34,116.73],[0.326866,-0.251271,-0.905673,-0.0988914],[0,-1,1,0],[9E+09,9E+09,9E+09,9E+09,9E+09,9E+09]], vmax, z20, tWeldGun;
		MoveL [[56.99,1626.55,-72.67],[0.410474,-0.275782,-0.84185,-0.216205],[0,0,1,0],[9E+09,9E+09,9E+09,9E+09,9E+09,9E+09]], vmax, z20, tWeldGun;
		ArcLStart [[49.28,1632.40,-74.45],[0.41046,-0.275749,-0.841871,-0.216193],[0,0,1,0],[9E+09,9E+09,9E+09,9E+09,9E+09,9E+09]], v10, seam13, weld13, fine, tWeldGun;
		ArcLEnd [[51.27,1632.00,-107.06],[0.410475,-0.275775,-0.841856,-0.216189],[0,0,1,0],[9E+09,9E+09,9E+09,9E+09,9E+09,9E+09]], v10, seam13, weld13, fine, tWeldGun;
		MoveL [[63.32,1618.59,53.83],[0.41045,-0.275792,-0.841833,-0.216304],[0,0,1,0],[9E+09,9E+09,9E+09,9E+09,9E+09,9E+09]], vmax, z20, tWeldGun;
		MoveJ [[774.48,1618.06,-14.91],[0.410442,-0.275748,-0.841846,-0.216328],[0,0,1,0],[9E+09,9E+09,9E+09,9E+09,9E+09,9E+09]], vmax, z20, tWeldGun;
		MoveL [[774.44,1618.01,-79.45],[0.410464,-0.275799,-0.841828,-0.216288],[0,0,0,0],[9E+09,9E+09,9E+09,9E+09,9E+09,9E+09]], vmax, z20, tWeldGun;
		ArcLStart [[760.64,1625.90,-79.46],[0.410464,-0.275804,-0.841826,-0.216291],[0,0,1,0],[9E+09,9E+09,9E+09,9E+09,9E+09,9E+09]], v10, seam13, weld13, fine, tWeldGun;
		ArcLEnd [[761.81,1625.90,-106.65],[0.410464,-0.2758,-0.841828,-0.216289],[0,0,1,0],[9E+09,9E+09,9E+09,9E+09,9E+09,9E+09]], v10, seam13, weld13, fine, tWeldGun;
		MoveL [[783.26,1604.44,251.05],[0.410482,-0.275804,-0.84182,-0.216279],[0,0,1,0],[9E+09,9E+09,9E+09,9E+09,9E+09,9E+09]], vmax, z20, tWeldGun;
		MoveJ pSafeS1, vmax, fine, tWeldGun;
	ENDPROC
	PROC ProSkid50()
		MoveJ [[314.39,1632.04,274.09],[0.410833,-0.611914,-0.675728,-0.0129978],[0,0,-3,0],[9E+09,9E+09,9E+09,9E+09,9E+09,9E+09]], vmax, z50, tWeldGun;
		MoveL [[314.32,1632.00,-25.30],[0.410826,-0.611972,-0.675681,-0.0129369],[0,0,-3,0],[9E+09,9E+09,9E+09,9E+09,9E+09,9E+09]], vmax, z50, tWeldGun;
		ArcLStart [[314.43,1633.11,-39.30],[0.349657,-0.639186,-0.683585,-0.0435139],[0,0,-3,0],[9E+09,9E+09,9E+09,9E+09,9E+09,9E+09]], v10, seam13, weld13, fine, tWeldGun;
		ArcL [[333.87,1632.50,-40.55],[0.349642,-0.639186,-0.683593,-0.0435083],[0,0,-3,0],[9E+09,9E+09,9E+09,9E+09,9E+09,9E+09]], v10, seam13, weld13, z5, tWeldGun;
		ArcL [[341.01,1631.27,-66.17],[0.317739,-0.654055,-0.683899,-0.0594762],[0,0,-3,0],[9E+09,9E+09,9E+09,9E+09,9E+09,9E+09]], v10, seam13, weld13, z5, tWeldGun;
		ArcLEnd [[358.67,1633.28,-65.92],[0.326244,-0.656849,-0.673963,-0.0888224],[0,0,-3,0],[9E+09,9E+09,9E+09,9E+09,9E+09,9E+09]], v10, seam13, weld13, fine, tWeldGun;
		MoveL [[364.49,1617.70,-14.89],[0.410824,-0.611946,-0.675708,-0.012893],[0,0,-3,0],[9E+09,9E+09,9E+09,9E+09,9E+09,9E+09]], vmax, z50, tWeldGun;
		MoveJ [[320.64,789.47,304.99],[0.235374,0.107276,-0.920325,0.293418],[0,-1,-4,0],[9E+09,9E+09,9E+09,9E+09,9E+09,9E+09]], vmax, z50, tWeldGun;
		MoveL [[320.65,680.04,-28.04],[0.235364,0.107285,-0.920324,0.293424],[0,-1,-4,0],[9E+09,9E+09,9E+09,9E+09,9E+09,9E+09]], vmax, z50, tWeldGun;
		ArcLStart [[320.49,676.84,-46.47],[0.235331,0.107401,-0.920274,0.293565],[0,-1,-4,0],[9E+09,9E+09,9E+09,9E+09,9E+09,9E+09]], v10, seam13, weld13, fine, tWeldGun;
		ArcL [[339.64,676.63,-48.64],[0.235361,0.107405,-0.920265,0.293567],[0,-1,-4,0],[9E+09,9E+09,9E+09,9E+09,9E+09,9E+09]], v5, seam13, weld13, z5, tWeldGun;
		ArcL [[342.53,676.66,-71.41],[0.281426,0.0897427,-0.912937,0.281589],[0,-1,-4,0],[9E+09,9E+09,9E+09,9E+09,9E+09,9E+09]], v5, seam13, weld13, z5, tWeldGun;
		ArcLEnd [[360.55,681.94,-73.50],[0.314989,0.316109,-0.866408,0.224044],[0,-1,-4,0],[9E+09,9E+09,9E+09,9E+09,9E+09,9E+09]], v10, seam13, weld13, fine, tWeldGun;
		MoveL [[365.60,682.37,3.04],[0.235347,0.107379,-0.920294,0.293497],[0,-1,-4,0],[9E+09,9E+09,9E+09,9E+09,9E+09,9E+09]], vmax, z50, tWeldGun;
		MoveJ [[836.02,763.37,35.73],[0.0217026,-0.41169,0.816455,-0.40428],[0,-2,-4,0],[9E+09,9E+09,9E+09,9E+09,9E+09,9E+09]], vmax, z50, tWeldGun;
		MoveL [[856.70,689.76,-27.01],[0.0217072,-0.411704,0.816444,-0.404287],[0,-2,-3,0],[9E+09,9E+09,9E+09,9E+09,9E+09,9E+09]], vmax, z50, tWeldGun;
		ArcLStart [[857.91,678.67,-44.98],[0.0203271,-0.414175,0.82252,-0.389238],[0,-2,-3,0],[9E+09,9E+09,9E+09,9E+09,9E+09,9E+09]], v10, seam13, weld13, fine, tWeldGun;
		ArcL [[836.15,679.48,-46.99],[0.0203132,-0.414191,0.822508,-0.389249],[0,-2,-3,0],[9E+09,9E+09,9E+09,9E+09,9E+09,9E+09]], v10, seam13, weld13, z5, tWeldGun;
		ArcL [[831.91,680.96,-69.65],[0.0726329,-0.437948,0.812132,-0.37864],[0,-2,-3,0],[9E+09,9E+09,9E+09,9E+09,9E+09,9E+09]], v10, seam13, weld13, z5, tWeldGun;
		ArcLEnd [[814.71,680.94,-69.65],[0.0726252,-0.437942,0.812135,-0.378643],[0,-2,-3,0],[9E+09,9E+09,9E+09,9E+09,9E+09,9E+09]], v10, seam13, weld13, fine, tWeldGun;
		MoveL [[809.35,725.26,127.04],[0.0216773,-0.411756,0.816405,-0.404315],[0,-2,-4,0],[9E+09,9E+09,9E+09,9E+09,9E+09,9E+09]], vmax, z50, tWeldGun;
		MoveJ [[841.70,1629.86,72.25],[0.220866,-0.864976,-0.348476,-0.285657],[0,0,-2,0],[9E+09,9E+09,9E+09,9E+09,9E+09,9E+09]], vmax, z50, tWeldGun;
		MoveL [[841.69,1629.87,-34.30],[0.220872,-0.864976,-0.348474,-0.285654],[0,0,-2,0],[9E+09,9E+09,9E+09,9E+09,9E+09,9E+09]], vmax, z50, tWeldGun;
		ArcLStart [[848.66,1634.80,-44.07],[0.220862,-0.865006,-0.348435,-0.28562],[0,0,-2,0],[9E+09,9E+09,9E+09,9E+09,9E+09,9E+09]], v20, seam13, weld13, fine, tWeldGun;
		ArcL [[827.08,1634.97,-46.50],[0.220852,-0.865009,-0.348428,-0.285626],[0,0,-2,0],[9E+09,9E+09,9E+09,9E+09,9E+09,9E+09]], v10, seam13, weld13, z1, tWeldGun;
		ArcL [[824.68,1632.91,-69.83],[0.143373,-0.869884,-0.317855,-0.348876],[0,0,-2,0],[9E+09,9E+09,9E+09,9E+09,9E+09,9E+09]], v10, seam13, weld13, z1, tWeldGun;
		ArcLEnd [[803.26,1635.12,-68.75],[0.265625,-0.855119,-0.383795,-0.225647],[0,0,-3,0],[9E+09,9E+09,9E+09,9E+09,9E+09,9E+09]], v10, seam13, weld13, fine, tWeldGun;
		MoveL [[798.38,1604.44,59.29],[0.220844,-0.86502,-0.348413,-0.285617],[0,0,-2,0],[9E+09,9E+09,9E+09,9E+09,9E+09,9E+09]], vmax, z50, tWeldGun;
		MoveJ [[1012.25,1627.55,26.24],[0.148022,-0.852995,-0.305302,-0.396586],[0,-1,-2,0],[9E+09,9E+09,9E+09,9E+09,9E+09,9E+09]], vmax, z50, tWeldGun;
		MoveL [[1012.25,1627.54,-29.96],[0.148013,-0.852994,-0.305304,-0.39659],[0,-1,-2,0],[9E+09,9E+09,9E+09,9E+09,9E+09,9E+09]], vmax, z50, tWeldGun;
		ArcLStart [[1020.33,1635.81,-42.74],[0.234694,-0.797645,-0.305793,-0.463867],[0,0,-2,0],[9E+09,9E+09,9E+09,9E+09,9E+09,9E+09]], v10, seam13, weld13, fine, tWeldGun;
		ArcLEnd [[1020.32,1636.60,-101.76],[0.234691,-0.797653,-0.305783,-0.463861],[0,0,-2,0],[9E+09,9E+09,9E+09,9E+09,9E+09,9E+09]], v10, seam13, weld13, fine, tWeldGun;
		MoveL [[1000.64,1624.71,1.80],[0.147993,-0.85301,-0.305288,-0.396575],[0,-1,-2,0],[9E+09,9E+09,9E+09,9E+09,9E+09,9E+09]], vmax, z50, tWeldGun;
		MoveJ [[999.85,699.71,74.25],[0.145952,0.855608,-0.347947,0.354353],[0,0,-2,0],[9E+09,9E+09,9E+09,9E+09,9E+09,9E+09]], vmax, z50, tWeldGun;
		MoveL [[1000.23,680.99,-33.60],[0.145957,0.855605,-0.347951,0.354355],[0,0,-2,0],[9E+09,9E+09,9E+09,9E+09,9E+09,9E+09]], vmax, z50, tWeldGun;
		ArcLStart [[1012.62,673.90,-46.78],[0.1719,0.826331,-0.335983,0.418023],[0,-1,-1,0],[9E+09,9E+09,9E+09,9E+09,9E+09,9E+09]], v10, seam13, weld13, fine, tWeldGun;
		ArcLEnd [[1014.09,670.24,-110.35],[0.203441,0.797575,-0.333295,0.459784],[0,-1,-1,0],[9E+09,9E+09,9E+09,9E+09,9E+09,9E+09]], v10, seam13, weld13, fine, tWeldGun;
		MoveL [[991.82,687.85,-113.61],[0.188232,0.8013,-0.32459,0.46597],[0,-1,-1,0],[9E+09,9E+09,9E+09,9E+09,9E+09,9E+09]], vmax, z50, tWeldGun;
		MoveL [[991.30,687.21,122.60],[0.188682,0.80133,-0.324494,0.465805],[0,-1,-1,0],[9E+09,9E+09,9E+09,9E+09,9E+09,9E+09]], vmax, z50, tWeldGun;
		MoveJ [[1353.61,686.57,-9.49],[0.257647,0.673939,-0.273385,0.636149],[0,-1,-1,0],[9E+09,9E+09,9E+09,9E+09,9E+09,9E+09]], vmax, z50, tWeldGun;
		MoveL [[1366.45,676.52,-47.24],[0.257646,0.673939,-0.273392,0.636147],[0,-1,-1,0],[9E+09,9E+09,9E+09,9E+09,9E+09,9E+09]], vmax, z50, tWeldGun;
		MoveL [[1385.74,669.35,-53.86],[0.230513,0.683708,-0.247774,0.646542],[0,-1,-1,0],[9E+09,9E+09,9E+09,9E+09,9E+09,9E+09]], vmax, z50, tWeldGun;
		ArcLStart [[1396.72,664.95,-53.87],[0.230521,0.683708,-0.247794,0.64653],[0,-1,-1,0],[9E+09,9E+09,9E+09,9E+09,9E+09,9E+09]], v10, seam13, weld13, fine, tWeldGun;
		ArcLEnd [[1395.51,665.99,-104.00],[0.221455,0.706537,-0.255943,0.621496],[0,-1,-1,0],[9E+09,9E+09,9E+09,9E+09,9E+09,9E+09]], v10, seam13, weld13, fine, tWeldGun;
		MoveL [[1331.35,694.89,21.64],[0.250476,0.690284,-0.28012,0.618307],[0,-1,-1,0],[9E+09,9E+09,9E+09,9E+09,9E+09,9E+09]], vmax, z50, tWeldGun;
		MoveJ [[1376.90,1623.22,41.45],[0.127213,-0.647245,-0.354873,-0.662538],[0,-1,-2,0],[9E+09,9E+09,9E+09,9E+09,9E+09,9E+09]], vmax, z50, tWeldGun;
		MoveL [[1376.90,1623.22,-50.53],[0.127212,-0.647239,-0.354892,-0.662534],[0,-1,-2,0],[9E+09,9E+09,9E+09,9E+09,9E+09,9E+09]], vmax, z50, tWeldGun;
		MoveL [[1397.45,1625.31,-50.53],[0.127209,-0.647235,-0.354904,-0.662533],[0,-1,-2,0],[9E+09,9E+09,9E+09,9E+09,9E+09,9E+09]], vmax, z50, tWeldGun;
		ArcLStart [[1408.53,1635.18,-50.45],[0.13106,-0.646617,-0.358565,-0.66041],[0,-1,-2,0],[9E+09,9E+09,9E+09,9E+09,9E+09,9E+09]], v10, seam13, weld13, fine, tWeldGun;
		ArcLEnd [[1408.03,1635.82,-99.67],[0.131146,-0.646603,-0.358564,-0.660407],[0,-1,-2,0],[9E+09,9E+09,9E+09,9E+09,9E+09,9E+09]], v10, seam13, weld13, fine, tWeldGun;
		MoveL [[1363.68,1613.53,-100.12],[0.126344,-0.650949,-0.356972,-0.657932],[0,-1,-2,0],[9E+09,9E+09,9E+09,9E+09,9E+09,9E+09]], vmax, z50, tWeldGun;
		MoveL [[1363.68,1613.52,239.17],[0.126341,-0.650966,-0.356946,-0.65793],[0,-1,-2,0],[9E+09,9E+09,9E+09,9E+09,9E+09,9E+09]], vmax, z50, tWeldGun;
		MoveJ [[1053.29,1631.94,67.33],[0.645571,-0.290399,-0.679976,-0.191155],[0,0,-4,0],[9E+09,9E+09,9E+09,9E+09,9E+09,9E+09]], vmax, z50, tWeldGun;
		MoveL [[1050.64,1634.55,-48.97],[0.636579,-0.309627,-0.673934,-0.211453],[0,0,-4,0],[9E+09,9E+09,9E+09,9E+09,9E+09,9E+09]], vmax, z50, tWeldGun;
		ArcLStart [[1024.87,1642.92,-50.56],[0.620533,-0.340261,-0.661431,-0.248335],[0,0,-4,0],[9E+09,9E+09,9E+09,9E+09,9E+09,9E+09]], v40, seam13, weld13, fine, tWeldGun;
		ArcLEnd [[1024.76,1640.88,-101.10],[0.608555,-0.344646,-0.672494,-0.242141],[0,0,-4,0],[9E+09,9E+09,9E+09,9E+09,9E+09,9E+09]], v10, seam13, weld13, fine, tWeldGun;
		MoveL [[1059.23,1614.28,-98.92],[0.62811,-0.294152,-0.696928,-0.18233],[0,0,-4,0],[9E+09,9E+09,9E+09,9E+09,9E+09,9E+09]], vmax, z50, tWeldGun;
		MoveL [[1059.23,1614.28,101.64],[0.628115,-0.294149,-0.696925,-0.182328],[0,0,-4,0],[9E+09,9E+09,9E+09,9E+09,9E+09,9E+09]], vmax, z50, tWeldGun;
		MoveJ [[1052.30,694.66,47.76],[0.644485,0.276131,-0.67942,0.216286],[0,-1,-5,0],[9E+09,9E+09,9E+09,9E+09,9E+09,9E+09]], vmax, z50, tWeldGun;
		MoveL [[1046.18,687.12,-54.58],[0.644485,0.276128,-0.679419,0.216291],[0,-1,-5,0],[9E+09,9E+09,9E+09,9E+09,9E+09,9E+09]], vmax, z50, tWeldGun;
		ArcLStart [[1016.59,670.93,-55.13],[0.641006,0.272426,-0.686489,0.208876],[0,-1,-5,0],[9E+09,9E+09,9E+09,9E+09,9E+09,9E+09]], v40, seam13, weld13, fine, tWeldGun;
		ArcLEnd [[1018.18,671.82,-104.69],[0.610333,0.278617,-0.715977,0.192985],[0,-1,-5,0],[9E+09,9E+09,9E+09,9E+09,9E+09,9E+09]], v10, seam13, weld13, fine, tWeldGun;
		MoveL [[1061.24,699.45,-98.70],[0.621239,0.282704,-0.701168,0.206166],[0,-1,-5,0],[9E+09,9E+09,9E+09,9E+09,9E+09,9E+09]], vmax, z50, tWeldGun;
		MoveL [[1054.68,728.71,93.69],[0.621244,0.28271,-0.701163,0.206161],[0,-1,-5,0],[9E+09,9E+09,9E+09,9E+09,9E+09,9E+09]], vmax, z50, tWeldGun;
		MoveJ pSafeS1, vmax, z50, tWeldGun;
	ENDPROC
	PROC ProSkid100()
		MoveJ [[1291.14,1401.40,237.11],[0.110665,-0.797291,0.0809156,-0.587821],[0,-1,-2,0],[9E+09,9E+09,9E+09,9E+09,9E+09,9E+09]], vmax, z50, tWeldGun;
		MoveL [[1375.22,1595.27,-52.82],[0.288027,-0.714876,-0.187844,-0.608858],[0,0,-3,0],[9E+09,9E+09,9E+09,9E+09,9E+09,9E+09]], vmax, z50, tWeldGun;
		ArcLStart [[1401.19,1605.13,-53.85],[0.288002,-0.715075,-0.187416,-0.608768],[0,0,-3,0],[9E+09,9E+09,9E+09,9E+09,9E+09,9E+09]], v40, seam13, weld13, fine, tWeldGun;
		ArcLEnd [[1398.73,1603.16,-97.27],[0.291491,-0.748178,-0.222798,-0.552834],[0,0,-3,0],[9E+09,9E+09,9E+09,9E+09,9E+09,9E+09]], v10, seam13, weld13, fine, tWeldGun;
		MoveL [[1364.33,1598.00,-103.67],[0.29149,-0.748144,-0.222826,-0.552868],[0,0,-3,0],[9E+09,9E+09,9E+09,9E+09,9E+09,9E+09]], vmax, z50, tWeldGun;
		MoveL [[1364.34,1597.99,108.74],[0.291485,-0.748128,-0.222876,-0.552873],[0,0,-3,0],[9E+09,9E+09,9E+09,9E+09,9E+09,9E+09]], vmax, z50, tWeldGun;
		MoveJ [[1362.85,671.57,209.86],[0.286582,0.681473,-0.261257,0.620653],[0,-1,-1,0],[9E+09,9E+09,9E+09,9E+09,9E+09,9E+09]], vmax, z50, tWeldGun;
		MoveL [[1362.83,671.44,-56.38],[0.286695,0.6814,-0.261216,0.620699],[0,-1,-1,0],[9E+09,9E+09,9E+09,9E+09,9E+09,9E+09]], vmax, z50, tWeldGun;
		ArcLStart [[1395.77,665.10,-57.82],[0.286611,0.681406,-0.26142,0.620645],[0,-1,-1,0],[9E+09,9E+09,9E+09,9E+09,9E+09,9E+09]], v40, seam13, weld13, fine, tWeldGun;
		ArcLEnd [[1394.43,667.22,-108.56],[0.265195,0.724641,-0.280093,0.571066],[0,-1,-1,0],[9E+09,9E+09,9E+09,9E+09,9E+09,9E+09]], v10, seam13, weld13, fine, tWeldGun;
		MoveL [[1359.52,678.30,-105.63],[0.265193,0.724636,-0.280059,0.57109],[0,-1,-1,0],[9E+09,9E+09,9E+09,9E+09,9E+09,9E+09]], vmax, z50, tWeldGun;
		MoveL [[1359.46,678.32,110.96],[0.265199,0.724649,-0.280131,0.571035],[0,-1,-1,0],[9E+09,9E+09,9E+09,9E+09,9E+09,9E+09]], vmax, z50, tWeldGun;
		MoveJ [[1044.44,682.04,140.05],[0.601349,0.276396,-0.690912,0.290906],[0,-1,-1,0],[9E+09,9E+09,9E+09,9E+09,9E+09,9E+09]], vmax, z50, tWeldGun;
		MoveL [[1044.44,682.04,-56.39],[0.601349,0.276385,-0.690916,0.290907],[0,-1,-1,0],[9E+09,9E+09,9E+09,9E+09,9E+09,9E+09]], vmax, z50, tWeldGun;
		ArcLStart [[1017.57,668.39,-58.10],[0.603558,0.271588,-0.6932,0.285364],[0,-1,-1,0],[9E+09,9E+09,9E+09,9E+09,9E+09,9E+09]], v40, seam13, weld13, fine, tWeldGun;
		ArcLEnd [[1019.45,669.58,-104.61],[0.590639,0.26522,-0.716441,0.259839],[0,-1,-1,0],[9E+09,9E+09,9E+09,9E+09,9E+09,9E+09]], v10, seam13, weld13, fine, tWeldGun;
		MoveL [[1053.53,682.10,-104.02],[0.581859,0.284263,-0.707585,0.282771],[0,-1,-1,0],[9E+09,9E+09,9E+09,9E+09,9E+09,9E+09]], vmax, z50, tWeldGun;
		MoveL [[1053.53,682.10,204.32],[0.581854,0.284262,-0.707586,0.282779],[0,-1,-1,0],[9E+09,9E+09,9E+09,9E+09,9E+09,9E+09]], vmax, z50, tWeldGun;
		MoveJ [[1060.34,1591.42,255.61],[0.587485,-0.309916,-0.701855,-0.25732],[0,0,0,0],[9E+09,9E+09,9E+09,9E+09,9E+09,9E+09]], vmax, z50, tWeldGun;
		MoveL [[1053.26,1597.30,-47.55],[0.593101,-0.251297,-0.715306,-0.270959],[0,0,0,0],[9E+09,9E+09,9E+09,9E+09,9E+09,9E+09]], vmax, z50, tWeldGun;
		ArcLStart [[1026.61,1608.02,-51.00],[0.610395,-0.281453,-0.687146,-0.275743],[0,0,0,0],[9E+09,9E+09,9E+09,9E+09,9E+09,9E+09]], v40, seam13, weld13, fine, tWeldGun;
		ArcLEnd [[1026.10,1606.98,-99.41],[0.589939,-0.305128,-0.703921,-0.251723],[0,0,0,0],[9E+09,9E+09,9E+09,9E+09,9E+09,9E+09]], v10, seam13, weld13, fine, tWeldGun;
		MoveL [[1060.35,1591.41,-99.10],[0.587476,-0.309917,-0.701859,-0.257327],[0,0,0,0],[9E+09,9E+09,9E+09,9E+09,9E+09,9E+09]], vmax, z50, tWeldGun;
		MoveL [[1060.34,1591.42,255.61],[0.587485,-0.309915,-0.701855,-0.25732],[0,0,0,0],[9E+09,9E+09,9E+09,9E+09,9E+09,9E+09]], vmax, z50, tWeldGun;
		SingArea\Wrist;
		MoveJ [[1013.97,1596.58,293.15],[0.294503,-0.721995,-0.258472,-0.57025],[0,-1,-2,0],[9E+09,9E+09,9E+09,9E+09,9E+09,9E+09]], vmax, z50, tWeldGun;
		MoveL [[1013.98,1596.59,-30.67],[0.294506,-0.721988,-0.258475,-0.570255],[0,-1,-2,0],[9E+09,9E+09,9E+09,9E+09,9E+09,9E+09]], vmax, z50, tWeldGun;
		ArcLStart [[1023.71,1603.83,-45.32],[0.294459,-0.722161,-0.258075,-0.570242],[0,-1,-2,0],[9E+09,9E+09,9E+09,9E+09,9E+09,9E+09]], v40, seam13, weld13, fine, tWeldGun;
		ArcLEnd [[1025.41,1604.13,-103.60],[0.29453,-0.721895,-0.258759,-0.570231],[0,-2,-1,0],[9E+09,9E+09,9E+09,9E+09,9E+09,9E+09]], v10, seam13, weld13, fine, tWeldGun;
		MoveL [[1013.24,1596.64,-103.54],[0.294541,-0.721861,-0.258796,-0.570252],[0,-2,-1,0],[9E+09,9E+09,9E+09,9E+09,9E+09,9E+09]], vmax, z50, tWeldGun;
		MoveL [[1013.24,1596.64,216.29],[0.294538,-0.721863,-0.258801,-0.570249],[0,-1,-2,0],[9E+09,9E+09,9E+09,9E+09,9E+09,9E+09]], vmax, z50, tWeldGun;
		MoveJ [[1006.20,679.01,292.67],[0.249851,0.680628,-0.312953,0.613499],[0,-1,-1,0],[9E+09,9E+09,9E+09,9E+09,9E+09,9E+09]], vmax, z50, tWeldGun;
		MoveL [[1006.17,679.00,-34.38],[0.24986,0.680635,-0.312969,0.61348],[0,-1,-1,0],[9E+09,9E+09,9E+09,9E+09,9E+09,9E+09]], vmax, z50, tWeldGun;
		ArcLStart [[1018.04,667.69,-51.11],[0.249871,0.680622,-0.312899,0.613525],[0,-1,-1,0],[9E+09,9E+09,9E+09,9E+09,9E+09,9E+09]], v40, seam13, weld13, fine, tWeldGun;
		ArcLEnd [[1018.17,669.74,-109.45],[0.216526,0.718194,-0.30883,0.584755],[0,-1,-1,0],[9E+09,9E+09,9E+09,9E+09,9E+09,9E+09]], v10, seam13, weld13, fine, tWeldGun;
		MoveL [[1006.90,676.88,-109.46],[0.216515,0.7182,-0.3088,0.584767],[0,-1,-1,0],[9E+09,9E+09,9E+09,9E+09,9E+09,9E+09]], vmax, z50, tWeldGun;
		MoveL [[1006.79,676.72,112.07],[0.216658,0.718018,-0.309197,0.584729],[0,-1,-1,0],[9E+09,9E+09,9E+09,9E+09,9E+09,9E+09]], vmax, z50, tWeldGun;
		MoveJ [[787.15,693.27,162.12],[0.200359,0.831329,-0.351726,0.38084],[0,-1,-1,0],[9E+09,9E+09,9E+09,9E+09,9E+09,9E+09]], vmax, z50, tWeldGun;
		MoveL [[803.22,683.52,-42.38],[0.200572,0.831304,-0.351703,0.380802],[0,-1,-1,0],[9E+09,9E+09,9E+09,9E+09,9E+09,9E+09]], vmax, z50, tWeldGun;
		ArcLStart [[820.10,672.81,-46.13],[0.200379,0.831311,-0.351741,0.380853],[0,-1,-1,0],[9E+09,9E+09,9E+09,9E+09,9E+09,9E+09]], v40, seam13, weld13, fine, tWeldGun;
		ArcL [[817.01,674.25,-61.57],[0.20037,0.83131,-0.351759,0.380844],[0,-1,-1,0],[9E+09,9E+09,9E+09,9E+09,9E+09,9E+09]], v5, seam13, weld13, z1, tWeldGun;
		ArcLEnd [[794.94,677.39,-61.37],[0.290522,0.768851,-0.506548,0.260529],[0,0,-1,0],[9E+09,9E+09,9E+09,9E+09,9E+09,9E+09]], v5, seam13, weld13, fine, tWeldGun;
		MoveL [[734.17,714.46,-10.08],[0.200543,0.831312,-0.351674,0.380825],[0,-1,-1,0],[9E+09,9E+09,9E+09,9E+09,9E+09,9E+09]], vmax, z50, tWeldGun;
		MoveJ [[728.25,1535.19,24.79],[0.147924,-0.86943,-0.34114,-0.325322],[0,0,-2,0],[9E+09,9E+09,9E+09,9E+09,9E+09,9E+09]], vmax, z50, tWeldGun;
		MoveL [[809.40,1591.07,-32.04],[0.147916,-0.869421,-0.341164,-0.325324],[0,0,-2,0],[9E+09,9E+09,9E+09,9E+09,9E+09,9E+09]], vmax, z50, tWeldGun;
		ArcLStart [[827.85,1598.76,-39.10],[0.147892,-0.869436,-0.341158,-0.325301],[0,0,-2,0],[9E+09,9E+09,9E+09,9E+09,9E+09,9E+09]], v40, seam13, weld13, fine, tWeldGun;
		ArcL [[824.60,1599.34,-54.56],[0.213243,-0.841559,-0.352486,-0.34937],[0,0,-2,0],[9E+09,9E+09,9E+09,9E+09,9E+09,9E+09]], v5, seam13, weld13, z1, tWeldGun;
		ArcLEnd [[804.61,1597.85,-55.38],[0.172397,-0.84314,-0.38332,-0.335351],[0,0,-2,0],[9E+09,9E+09,9E+09,9E+09,9E+09,9E+09]], v5, seam13, weld13, fine, tWeldGun;
		MoveL [[776.91,1584.46,5.55],[0.169992,-0.855201,-0.338248,-0.354009],[0,0,-2,0],[9E+09,9E+09,9E+09,9E+09,9E+09,9E+09]], vmax, z50, tWeldGun;
		MoveJ [[190.08,1566.54,31.00],[0.344053,-0.456867,-0.796918,-0.19448],[0,0,1,0],[9E+09,9E+09,9E+09,9E+09,9E+09,9E+09]], vmax, z50, tWeldGun;
		MoveL [[140.48,1600.64,-31.65],[0.344036,-0.456857,-0.79694,-0.194443],[0,0,1,0],[9E+09,9E+09,9E+09,9E+09,9E+09,9E+09]], vmax, z50, tWeldGun;
		ArcLStart [[132.97,1606.81,-38.27],[0.398419,-0.43769,-0.785543,-0.180589],[0,0,1,0],[9E+09,9E+09,9E+09,9E+09,9E+09,9E+09]], v40, seam13, weld13, fine, tWeldGun;
		ArcL [[137.87,1603.07,-53.48],[0.330333,-0.450337,-0.806737,-0.19301],[0,-1,1,0],[9E+09,9E+09,9E+09,9E+09,9E+09,9E+09]], v5, seam13, weld13, z1, tWeldGun;
		ArcLEnd [[160.89,1601.52,-53.60],[0.247106,-0.517365,-0.784142,-0.237474],[0,-1,1,0],[9E+09,9E+09,9E+09,9E+09,9E+09,9E+09]], v5, seam13, weld13, fine, tWeldGun;
		MoveL [[175.52,1584.51,-47.94],[0.344043,-0.456835,-0.796927,-0.194535],[0,0,1,0],[9E+09,9E+09,9E+09,9E+09,9E+09,9E+09]], vmax, z50, tWeldGun;
		MoveJ [[182.42,764.05,86.85],[0.357832,0.377008,-0.841375,0.14802],[0,0,0,0],[9E+09,9E+09,9E+09,9E+09,9E+09,9E+09]], vmax, z50, tWeldGun;
		MoveL [[138.47,690.39,-38.58],[0.357921,0.376925,-0.841359,0.148106],[0,0,0,0],[9E+09,9E+09,9E+09,9E+09,9E+09,9E+09]], vmax, z50, tWeldGun;
		ArcLStart [[127.27,682.76,-39.17],[0.357916,0.376949,-0.841354,0.148087],[0,0,0,0],[9E+09,9E+09,9E+09,9E+09,9E+09,9E+09]], v40, seam13, weld13, fine, tWeldGun;
		ArcL [[131.33,682.78,-57.87],[0.357887,0.376962,-0.841374,0.148009],[0,0,0,0],[9E+09,9E+09,9E+09,9E+09,9E+09,9E+09]], v5, seam13, weld13, z1, tWeldGun;
		ArcLEnd [[152.38,682.50,-58.95],[0.357948,0.376909,-0.841357,0.148091],[0,0,0,0],[9E+09,9E+09,9E+09,9E+09,9E+09,9E+09]], v5, seam13, weld13, fine, tWeldGun;
		MoveL [[182.36,703.78,23.74],[0.357926,0.376967,-0.841339,0.1481],[0,0,0,0],[9E+09,9E+09,9E+09,9E+09,9E+09,9E+09]], vmax, z50, tWeldGun;
		MoveJ [[104.88,808.11,108.60],[0.181133,-0.65989,-0.702536,-0.195398],[0,-1,1,0],[9E+09,9E+09,9E+09,9E+09,9E+09,9E+09]], vmax, z50, tWeldGun;
		MoveL [[104.87,808.11,-22.73],[0.181133,-0.6599,-0.702527,-0.195398],[0,-1,1,0],[9E+09,9E+09,9E+09,9E+09,9E+09,9E+09]], vmax, z50, tWeldGun;
		ArcLStart [[104.88,808.11,-33.52],[0.181134,-0.659877,-0.702547,-0.1954],[0,-1,1,0],[9E+09,9E+09,9E+09,9E+09,9E+09,9E+09]], v10, seam13, weld13, fine, tWeldGun;
		ArcLEnd [[119.95,808.11,-33.52],[0.181133,-0.659872,-0.702552,-0.195399],[0,-1,1,0],[9E+09,9E+09,9E+09,9E+09,9E+09,9E+09]], v10, seam13, weld13, fine, tWeldGun;
		MoveL [[119.95,808.11,110.38],[0.181135,-0.659885,-0.70254,-0.1954],[0,-1,1,0],[9E+09,9E+09,9E+09,9E+09,9E+09,9E+09]], vmax, z50, tWeldGun;
		MoveJ [[104.20,866.55,110.15],[0.247858,0.624252,-0.690017,0.269727],[0,-1,0,0],[9E+09,9E+09,9E+09,9E+09,9E+09,9E+09]], vmax, z50, tWeldGun;
		MoveL [[104.20,866.56,-18.99],[0.247849,0.624251,-0.690021,0.269728],[0,-1,0,0],[9E+09,9E+09,9E+09,9E+09,9E+09,9E+09]], vmax, z50, tWeldGun;
		ArcLStart [[104.22,866.56,-33.89],[0.247832,0.624264,-0.690012,0.269738],[0,-1,0,0],[9E+09,9E+09,9E+09,9E+09,9E+09,9E+09]], v10, seam13, weld13, fine, tWeldGun;
		ArcLEnd [[117.44,866.46,-33.99],[0.247835,0.624263,-0.690014,0.269732],[0,-1,0,0],[9E+09,9E+09,9E+09,9E+09,9E+09,9E+09]], v10, seam13, weld13, fine, tWeldGun;
		MoveL [[117.44,866.45,125.28],[0.247841,0.62426,-0.690014,0.269731],[0,-1,0,0],[9E+09,9E+09,9E+09,9E+09,9E+09,9E+09]], vmax, z50, tWeldGun;
		MoveJ [[108.37,1419.35,200.82],[0.287761,-0.638557,-0.653225,-0.28764],[0,-1,1,0],[9E+09,9E+09,9E+09,9E+09,9E+09,9E+09]], vmax, z50, tWeldGun;
		MoveL [[109.57,1420.53,-14.32],[0.263504,-0.648771,-0.662871,-0.265072],[0,-1,1,0],[9E+09,9E+09,9E+09,9E+09,9E+09,9E+09]], vmax, z50, tWeldGun;
		ArcLStart [[109.57,1420.55,-29.31],[0.263511,-0.648758,-0.662878,-0.26508],[0,-1,1,0],[9E+09,9E+09,9E+09,9E+09,9E+09,9E+09]], v10, seam13, weld13, fine, tWeldGun;
		ArcLEnd [[121.97,1420.55,-29.31],[0.26351,-0.648759,-0.662878,-0.265081],[0,-1,1,0],[9E+09,9E+09,9E+09,9E+09,9E+09,9E+09]], v10, seam13, weld13, fine, tWeldGun;
		MoveL [[121.96,1420.55,113.82],[0.263512,-0.648767,-0.662871,-0.265077],[0,-1,1,0],[9E+09,9E+09,9E+09,9E+09,9E+09,9E+09]], vmax, z50, tWeldGun;
		MoveJ [[107.74,1476.86,132.75],[0.227381,0.67854,-0.65675,0.237825],[0,0,-1,0],[9E+09,9E+09,9E+09,9E+09,9E+09,9E+09]], vmax, z50, tWeldGun;
		MoveL [[107.75,1476.86,-6.53],[0.227369,0.678545,-0.656746,0.237835],[0,0,-1,0],[9E+09,9E+09,9E+09,9E+09,9E+09,9E+09]], vmax, z50, tWeldGun;
		ArcLStart [[105.63,1476.40,-27.57],[0.227388,0.678538,-0.656756,0.237808],[0,0,-1,0],[9E+09,9E+09,9E+09,9E+09,9E+09,9E+09]], v40, seam13, weld13, fine, tWeldGun;
		ArcLEnd [[119.62,1476.10,-27.13],[0.227387,0.678539,-0.656755,0.237809],[0,0,-1,0],[9E+09,9E+09,9E+09,9E+09,9E+09,9E+09]], v10, seam13, weld13, fine, tWeldGun;
		MoveL [[118.38,1476.85,2.29],[0.227385,0.678544,-0.656744,0.237828],[0,0,-1,0],[9E+09,9E+09,9E+09,9E+09,9E+09,9E+09]], vmax, z50, tWeldGun;
		MoveL [[836.49,1471.77,-21.22],[0.227415,0.678515,-0.656775,0.237796],[0,0,-1,0],[9E+09,9E+09,9E+09,9E+09,9E+09,9E+09]], vmax, z50, tWeldGun;
		ArcLStart [[833.70,1470.86,-31.25],[0.227422,0.678532,-0.656755,0.237797],[0,0,-1,0],[9E+09,9E+09,9E+09,9E+09,9E+09,9E+09]], v10, seam13, weld13, fine, tWeldGun;
		ArcLEnd [[848.24,1470.72,-30.35],[0.227417,0.67853,-0.656757,0.2378],[0,0,-1,0],[9E+09,9E+09,9E+09,9E+09,9E+09,9E+09]], v10, seam13, weld13, fine, tWeldGun;
		MoveL [[845.94,1471.75,199.33],[0.227429,0.678527,-0.65675,0.237818],[0,0,-1,0],[9E+09,9E+09,9E+09,9E+09,9E+09,9E+09]], vmax, z50, tWeldGun;
		MoveJ [[851.82,1398.82,138.77],[0.249585,-0.660425,-0.662158,-0.251183],[0,-1,1,0],[9E+09,9E+09,9E+09,9E+09,9E+09,9E+09]], vmax, z50, tWeldGun;
		MoveL [[851.80,1413.16,-17.04],[0.24959,-0.660434,-0.662152,-0.251173],[0,-1,1,0],[9E+09,9E+09,9E+09,9E+09,9E+09,9E+09]], vmax, z50, tWeldGun;
		ArcLStart [[851.81,1413.17,-30.35],[0.249586,-0.660427,-0.662156,-0.251181],[0,-1,1,0],[9E+09,9E+09,9E+09,9E+09,9E+09,9E+09]], v40, seam13, weld13, fine, tWeldGun;
		ArcLEnd [[837.71,1413.17,-30.35],[0.249589,-0.660431,-0.662154,-0.251176],[0,-1,1,0],[9E+09,9E+09,9E+09,9E+09,9E+09,9E+09]], v10, seam13, weld13, fine, tWeldGun;
		MoveL [[837.70,1413.16,114.72],[0.24959,-0.660435,-0.662151,-0.251172],[0,-1,1,0],[9E+09,9E+09,9E+09,9E+09,9E+09,9E+09]], vmax, z50, tWeldGun;
		MoveJ [[836.86,863.49,66.47],[0.245499,0.671633,-0.652073,0.251873],[0,0,-1,0],[9E+09,9E+09,9E+09,9E+09,9E+09,9E+09]], vmax, z50, tWeldGun;
		MoveL [[833.18,862.81,-20.93],[0.245535,0.671618,-0.652081,0.251858],[0,0,-1,0],[9E+09,9E+09,9E+09,9E+09,9E+09,9E+09]], vmax, z50, tWeldGun;
		ArcLStart [[832.14,861.68,-36.34],[0.245527,0.671615,-0.652094,0.25184],[0,0,-1,0],[9E+09,9E+09,9E+09,9E+09,9E+09,9E+09]], v40, seam13, weld13, fine, tWeldGun;
		ArcLEnd [[847.39,860.80,-37.23],[0.245547,0.671614,-0.652088,0.251841],[0,0,-1,0],[9E+09,9E+09,9E+09,9E+09,9E+09,9E+09]], v10, seam13, weld13, fine, tWeldGun;
		MoveL [[844.19,862.64,90.70],[0.24553,0.671618,-0.652082,0.251861],[0,0,-1,0],[9E+09,9E+09,9E+09,9E+09,9E+09,9E+09]], vmax, z50, tWeldGun;
		MoveJ [[850.02,796.71,104.60],[0.232706,-0.667694,-0.66755,-0.23326],[0,-1,1,0],[9E+09,9E+09,9E+09,9E+09,9E+09,9E+09]], vmax, z50, tWeldGun;
		MoveL [[848.57,804.07,-20.25],[0.232717,-0.667711,-0.667535,-0.233244],[0,-1,1,0],[9E+09,9E+09,9E+09,9E+09,9E+09,9E+09]], vmax, z50, tWeldGun;
		ArcLStart [[848.57,804.08,-35.68],[0.232715,-0.667709,-0.667535,-0.233251],[0,-1,1,0],[9E+09,9E+09,9E+09,9E+09,9E+09,9E+09]], v40, seam13, weld13, fine, tWeldGun;
		ArcLEnd [[836.56,803.94,-35.91],[0.232718,-0.667714,-0.66753,-0.233248],[0,-1,1,0],[9E+09,9E+09,9E+09,9E+09,9E+09,9E+09]], v10, seam13, weld13, fine, tWeldGun;
		MoveL [[836.55,803.93,282.92],[0.232721,-0.66772,-0.667527,-0.233237],[0,-1,1,0],[9E+09,9E+09,9E+09,9E+09,9E+09,9E+09]], vmax, z50, tWeldGun;
		MoveJ pSafeS1, vmax, z50, tWeldGun;
	ENDPROC
ENDMODULE
